// TIA Portal V19 export
// export: Created 2026-08-20T21:47:30.4170897Z, ExportSetting WithDefaults, DisplayName Totally Integrated Automation Portal, DisplayVersion V19, DisplayName TIA Portal Openness, DisplayVersion V19, DisplayName TIA Portal Version Control Interface, DisplayVersion V19, DisplayName STEP 7 Professional, DisplayVersion V19, DisplayName STEP 7 Safety, DisplayVersion V19, DisplayName WinCC Basic/Comfort/Advanced, DisplayVersion V19, DisplayName WinCC Unified, DisplayVersion V19
FUNCTION_BLOCK "FB_SafetyPermissives"   // FB2, SCL
{ S7_Optimized_Access := 'TRUE' }
VERSION : 0.1
// Interlocks and alarms; runs every scan.
//  generated by LADDER - do not edit by hand
// stored: AutoNumber true, IsIECCheckEnabled false, IsRetainMemResEnabled false, MemoryReserve 100, SetENOAutomatically false, UDAEnableTagReadback false
   VAR
      IL_shutter_rst_mem : Bool;   // edge memory for reset_pb
      ALM_vacuum_ton { S7_SetPoint := 'True'} : TON_TIME;   // on-delay for alarm ALM_vacuum
      ALM_vacuum_ack_mem : Bool;   // edge memory for ack_pb
      ALM_pump_fb_ton { S7_SetPoint := 'True'} : TON_TIME;   // on-delay for alarm ALM_pump_fb
      ALM_pump_fb_ack_mem : Bool;   // edge memory for ack_pb
   END_VAR
BEGIN
       // interlock IL_shutter: Beam shutter permissive - trips on vacuum or valve fault.
       IF NOT ("pressure_ok" AND "gate_valve_closed") THEN
           "beam_shutter_permit" := FALSE;
       END_IF;
       IF "reset_pb" AND NOT #IL_shutter_rst_mem AND ("pressure_ok" AND "gate_valve_closed") THEN
           "beam_shutter_permit" := TRUE;
       END_IF;
       #IL_shutter_rst_mem := "reset_pb";
       // alarm [critical] ALM_vacuum: Vacuum lost (debounced 2 s), latched until acknowledged.
       #ALM_vacuum_ton(IN := NOT "pressure_ok",
                       PT := T#2s);
       IF #ALM_vacuum_ton.Q THEN
           "vacuum_alarm" := TRUE;
       END_IF;
       IF "ack_pb" AND NOT #ALM_vacuum_ack_mem AND NOT #ALM_vacuum_ton.Q THEN
           "vacuum_alarm" := FALSE;
       END_IF;
       #ALM_vacuum_ack_mem := "ack_pb";
       // alarm [alarm] ALM_pump_fb: Pump commanded but no running feedback within 5 s.
       #ALM_pump_fb_ton(IN := "pump_start_cmd" AND NOT "pump_running_fb",
                        PT := T#5s);
       IF #ALM_pump_fb_ton.Q THEN
           "pump_fault_alarm" := TRUE;
       END_IF;
       IF "ack_pb" AND NOT #ALM_pump_fb_ack_mem AND NOT #ALM_pump_fb_ton.Q THEN
           "pump_fault_alarm" := FALSE;
       END_IF;
       #ALM_pump_fb_ack_mem := "ack_pb";
END_FUNCTION_BLOCK
